TYPE ST_Identity_PK3_OUT3 :
STRUCT
	ID	:STRING;
	ReadQuality:STRING;
END_STRUCT
END_TYPE

(* stored: Version 1.1.0.1, ProductVersion 3.1.4024.13
   DUT ST_Identity_PK3_OUT3: Id {eb30dd5c-baca-4c66-a553-630211daa047} *)
